TYPE ST_Auto_LowerFeedInConveyorStatus EXTENDS ST_StatusBasic :
STRUCT
END_STRUCT
END_TYPE

(* stored: Version 1.1.0.1, ProductVersion 3.1.4024.13
   DUT ST_Auto_LowerFeedInConveyorStatus: Id {d02a7903-6a24-4cba-be9a-505f6e4c89fd} *)
